Universal Robots PolyScope program: g01_nut_dropoff.urp

Program g01_nut_dropoff (installation=default directory=/programs createdIn=5.9.1.1031110 lastSavedIn=5.9.1.1031110 robotSerialNumber=20195501059)
Calibrated DH parameters: a=[0.000146, -0.418764, -0.053981, 0.000058, -0.000023, 0]; d=[0.162545, 37.319448, -206.067439, 168.881546, 0.09955, 0.099464]; alpha=[1.57004, -0.001979, 0.002304, 1.570607, -1.57066, 0]; deltaTheta=[0, -0.174616, -1.258233, 1.432844, -0.000001, 0]
Robot Program (runOnlyOnce=false)
  URCap Grip Check (Robotiq_Grippers, Robotiq Inc.) dataModel(ObjectDetectedKey=true, DimensionValidationKey=false, DimensionKey=100.0, DimensionDimensionPositiveGapKey=5.0, DimensionNegativeGapKey=5.0, GripperIdKey=1, ModelDefinedKey=true); state(isChildrenLocked=true)
    URCap If (Robotiq_Grippers, Robotiq Inc.)
      MoveL speed 250 mm/s, acceleration 1200 mm/s^2 (useActiveTCP=true) feature=Base
        Waypoint Waypoint (Variable): variable(featureName=g01_nut_pickup)
        MoveDirectionNode (selectedDirection=ZPlus toolParams=0.02, 1.2) feature=Joint_6_name
          Until TOOL_CONTACT_DETECTION (allowActions=true retraction=0 decelerationAcceleration=1 decelerationAngularAcceleration=34.906585)
            URCap Gripper (Robotiq_Grippers, Robotiq Inc.) dataModel(position=59.29411764705882, force=100.0, speed=100.0, positionInDouble=59.29411764705882, forceInDouble=100.0, speedInDouble=100.0, slaveIds=[9], blocking=true)
        Waypoint Waypoint (Variable): variable(featureName=g01_nut_pickup)
